(* IEC 61131-3 sources: xPLCCore/codesys_code/AxisGroupManager(FB), 4 files *)

(* ---- AxisGroupManager.st ---- *)
//==============================================================================
// Main Function Block Definition
//==============================================================================
FUNCTION_BLOCK AxisGroupManager

VAR
    // --- Internal State & Events ---
    _preState : E_RobotState := E_RobotState.NULL;
    _eState : E_RobotState := E_RobotState.NULL;
    _nxtState : E_RobotState := E_RobotState.NULL;

    _eCurrentEvent : E_RobotEvent := E_RobotEvent.EV_NONE; // Holds the event to be processed

    // --- Axis Configuration ---
    _agAxisGroup : REFERENCE TO AXIS_GROUP_REF_SM3; // Internal reference to the axis group

    // --- Status & Error Info ---
    _bIsHomed : BOOL;
    _bIsInError : BOOL;
    _dwErrorID : DWORD;
    _bReadyForOperation : BOOL;

    // --- Motion Control Function Blocks ---
    _fbPower : MC_Power;
    _fbGroupEnable : MC_GroupEnable;
    _fbGroupReset : MC_GroupReset;
    _fbGroupDisable : MC_GroupDisable;
    _fbHome : MC_Home;

	fbPowerReel   : MC_Power;
    fbResetReel   : MC_Reset;
    bReelPowerReq : BOOL; // Flag to request power for the reel motor
	SMC_GroupPower_0:SM3_Robotics.SMC_GroupPower;
	GroupPower_Flag:BOOL:=FALSE;
	//SMC_GroupReset_0:SM3_Robotics.MC_GroupReset;
	SMC_GroupDisable:SM3_Robotics.MC_GroupDisable;

	SMC_GroupReset:SM3_Robotics.MC_GroupReset;

	enable_fb:SM3_Robotics.MC_GroupEnable;

	homing_fb:FB_Homing;

	MoveLinearAbsolute_0: SM3_Robotics.MC_MoveLinearAbsolute;
	motionPoseRunPass:INT;
	motionPoseIdx:INT;

	stateCD:INT;

END_VAR

(* ---- FB_init.st ---- *)
//==============================================================================
// FB_init: Called once on startup to configure the FB instance.
//==============================================================================
METHOD FB_init : BOOL
VAR_INPUT
    bInitRetains : BOOL; // This parameter is required by the compiler
    bInCopyCode : BOOL;  // This parameter is required by the compiler

    // The robot's axis group
    agAxisGroup : REFERENCE TO AXIS_GROUP_REF_SM3;

END_VAR
VAR
    i : UINT;
END_VAR

// Store the reference to the axis group
_agAxisGroup REF= agAxisGroup;

FB_init := TRUE;

_eState:=E_RobotState.NULL;
_nxtState:=E_RobotState.UnInited;
Update(1);//exit old state
_preState:=_eState;
_eState:=_nxtState;
Update(-1);//enter new state

(* ---- Transition.st ---- *)
METHOD Transition : BOOL
VAR_INPUT
    eEvent : E_RobotEvent;
END_VAR
VAR_OUTPUT
	error:BOOL;
	new_state:E_RobotState;
END_VAR

new_state:=_eState;
CASE _eState OF
	E_RobotState.UnInited:
		CASE eEvent OF
			E_RobotEvent.EV_POWER_ON:
			 new_state:=E_RobotState.Powering;
		END_CASE

	E_RobotState.Powering:
		CASE eEvent OF
			E_RobotEvent.EV_POWER_OFF,
			E_RobotEvent.EV_ERROR,
			E_RobotEvent.EV_RESET:
			   new_state:=E_RobotState.UnInited;
			E_RobotEvent.EV_OK:
			   new_state:=E_RobotState.Powered;
		END_CASE
	E_RobotState.Powered:
		CASE eEvent OF
		E_RobotEvent.EV_GROUP_ENABLE:
			 new_state:=E_RobotState.GroupEnabling;
		END_CASE

	E_RobotState.GroupEnabling:
		CASE eEvent OF
		E_RobotEvent.EV_OK:
			 new_state:=E_RobotState.GroupEnabled;
		END_CASE

	E_RobotState.GroupEnabled:
		CASE eEvent OF
		E_RobotEvent.EV_HOME_GO:
			 new_state:=E_RobotState.Homing;
		E_RobotEvent.EV_HOME_GO_FORCE_SKIP:
			 new_state:=E_RobotState.Ready;
		END_CASE
	E_RobotState.Homing:
		CASE eEvent OF
		E_RobotEvent.EV_OK:
			 new_state:=E_RobotState.Ready;
		END_CASE

	E_RobotState.Ready:
		CASE eEvent OF
		E_RobotEvent.EV_HOME_GO:
			 new_state:=E_RobotState.Homing;
		END_CASE

	E_RobotState.Error:
		CASE eEvent OF
		E_RobotEvent.EV_RESET:
			 new_state:=E_RobotState.UnInited;
		END_CASE

END_CASE

IF(new_state=_eState)THEN//error/stop handling
	IF(eEvent=E_RobotEvent.EV_ERROR)THEN
		new_state:=E_RobotState.Error;
	END_IF

END_IF

IF(new_state<>_eState)THEN
  _nxtState:=new_state;
  Update(1);//exit old state
  _preState:=_eState;
  _eState:=_nxtState;
  Update(-1);//enter new state

END_IF

(* ---- Update.st ---- *)
METHOD Update : BOOL
VAR_INPUT
	//-1 enter, 0 update,1 exit current(_eState) state
	uidx:INT:=0;
END_VAR
VAR

END_VAR

Update:=TRUE;

CASE _eState OF
    E_RobotState.UnInited:
        IF(uidx=-1)THEN // On Entry
            GroupPower_Flag := FALSE;
            bReelPowerReq   := FALSE; // Single Axis Power Flag

            // Reset Group FBs
            SMC_GroupDisable(AxisGroup:=_agAxisGroup, Execute:=FALSE);
            SMC_GroupReset(AxisGroup:=_agAxisGroup, Execute:=FALSE);

            // Reset Single Axis FBs
            fbResetReel(Axis:= reelpullmotor, Execute:=FALSE);

            IoConfig_Globals.EtherCAT_Master_SoftMotion.xRestart:=TRUE;
        END_IF

        IF(uidx=0)THEN // On Update
            SMC_GroupDisable(AxisGroup:=_agAxisGroup, Execute:=TRUE);
            SMC_GroupReset(AxisGroup:=_agAxisGroup, Execute:=TRUE);

            // Reset the single motor
            fbResetReel(Axis:= reelpullmotor, Execute:=TRUE);

            IoConfig_Globals.EtherCAT_Master_SoftMotion();
            IoConfig_Globals.EtherCAT_Master_SoftMotion.xRestart:=FALSE;
        END_IF
        RETURN;

    E_RobotState.Powering:
        IF(uidx=-1)THEN
            GroupPower_Flag := FALSE;
            bReelPowerReq   := FALSE;
        ELSIF(uidx=0)THEN
            GroupPower_Flag := TRUE;
            bReelPowerReq   := TRUE;

            // Wait for BOTH the group and the reel motor to report powered
            IF(SMC_GroupPower_0.Status AND fbPowerReel.Status) THEN
                Transition(E_RobotEvent.EV_OK);
            ELSIF(SMC_GroupPower_0.Error OR fbPowerReel.Error) THEN
                Transition(E_RobotEvent.EV_ERROR);
            END_IF
        END_IF

    E_RobotState.Powered:
        IF(uidx=-1)THEN
            GroupPower_Flag := TRUE;
            bReelPowerReq   := TRUE;
        ELSIF(uidx=0)THEN
            // Keep both drives alive while waiting for group enable command
            GroupPower_Flag := TRUE;
            bReelPowerReq   := TRUE;
            IF(SMC_GroupPower_0.Error OR fbPowerReel.Error) THEN
                Transition(E_RobotEvent.EV_ERROR);
            END_IF
        END_IF

    E_RobotState.GroupEnabling:
        IF(uidx=-1)THEN
            enable_fb(AxisGroup:=_agAxisGroup, Execute:=FALSE);
        ELSIF(uidx=0)THEN
            enable_fb(AxisGroup:=_agAxisGroup, Execute:=TRUE);

            // Single motor is already enabled via MC_Power in previous state
            IF(enable_fb.Done) THEN
                Transition(E_RobotEvent.EV_OK);
            ELSIF(enable_fb.Error) THEN
                Transition(E_RobotEvent.EV_ERROR);
            END_IF
        END_IF

    E_RobotState.GroupEnabled:
        IF(uidx=-1)THEN
            GroupPower_Flag := TRUE;
            bReelPowerReq   := TRUE;
        ELSIF(uidx=0)THEN
            // Group is enabled, keep power asserted for normal operation
            GroupPower_Flag := TRUE;
            bReelPowerReq   := TRUE;
            IF(SMC_GroupPower_0.Error OR fbPowerReel.Error) THEN
                Transition(E_RobotEvent.EV_ERROR);
            END_IF
        END_IF

    E_RobotState.Homing:
        IF(uidx=-1)THEN
            homing_fb(bExecute:=FALSE);
            stateCD:=100;
        ELSIF(uidx=0)THEN
            GroupPower_Flag := TRUE;
            bReelPowerReq   := TRUE;
            homing_fb(bExecute:=TRUE);
            IF(homing_fb.bDone) THEN
                stateCD:=stateCD-1;
                IF(stateCD=0)THEN
                    Transition(E_RobotEvent.EV_OK);
                END_IF
            ELSIF(homing_fb.bError)THEN
                Transition(E_RobotEvent.EV_ERROR);
            ELSE
                stateCD:=100;
            END_IF
        ELSIF(uidx=1)THEN
            homing_fb(bExecute:=FALSE);
        END_IF

    E_RobotState.Ready:
        IF(uidx=-1)THEN
            GroupPower_Flag := TRUE;
            bReelPowerReq   := TRUE;
        ELSIF(uidx=0)THEN
            GroupPower_Flag := TRUE;
            bReelPowerReq   := TRUE;
            IF(SMC_GroupPower_0.Error OR fbPowerReel.Error) THEN
                Transition(E_RobotEvent.EV_ERROR);
            END_IF
        END_IF

    E_RobotState.Error:
        IF(uidx=-1)THEN
            GroupPower_Flag := FALSE;
            bReelPowerReq   := FALSE;

            SMC_GroupDisable(AxisGroup:=_agAxisGroup, Execute:=FALSE);
            SMC_GroupReset(AxisGroup:=_agAxisGroup, Execute:=FALSE);
            fbResetReel(Axis:= reelpullmotor, Execute:=FALSE);
        END_IF

        IF(uidx=0)THEN
            // Hold power commands low every scan while in Error
            GroupPower_Flag := FALSE;
            bReelPowerReq   := FALSE;
            SMC_GroupDisable(AxisGroup:=_agAxisGroup, Execute:=TRUE);
            SMC_GroupReset(AxisGroup:=_agAxisGroup, Execute:=TRUE);
            fbResetReel(Axis:= reelpullmotor, Execute:=TRUE);
        END_IF
END_CASE

// --- CALL FUNCTION BLOCKS OUTSIDE THE CASE ---

// 1. Robot Group Power
SMC_GroupPower_0(
    AxisGroup    := _agAxisGroup,
    Enable       := TRUE,
    bRegulatorOn := GroupPower_Flag,
    bDriveStart  := GroupPower_Flag
);

// 2. Single Motor Power (Reel Pull)
fbPowerReel(
    Axis         := reelpullmotor,
    Enable       := bReelPowerReq,
    bRegulatorOn := bReelPowerReq,
    bDriveStart  := bReelPowerReq
);

// 3. Single Motor Reset
fbResetReel(Axis := reelpullmotor);
